ABB RAPID module: Module1.mod

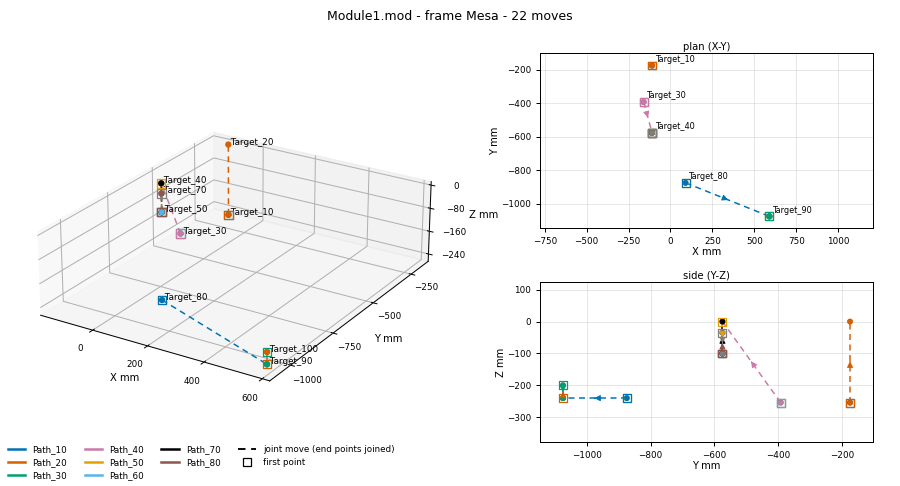
[picture p0: tool path of Module1.mod in frame Mesa, 22 of 23 moves have a stored position in this frame; points joined in program order, loops and branches not executed]
MODULE Module1
    CONST robtarget Target_10:=[[-110,-175,-254],[0.990340804,0,0,-0.138654579],[0,-2,0,0],[9E+09,9E+09,9E+09,9E+09,9E+09,9E+09]];
    CONST robtarget Target_20:=[[-110,-175,0],[0.990340804,0,0,-0.138654579],[0,-2,0,0],[9E+09,9E+09,9E+09,9E+09,9E+09,9E+09]];
    CONST robtarget Target_30:=[[-160,-392.5,-253.927],[1,0,0,0],[0,-2,0,0],[9E+09,9E+09,9E+09,9E+09,9E+09,9E+09]];
    CONST robtarget Target_40:=[[-110,-575,0],[0.990340804,0,0,0.138654579],[0,-2,0,0],[9E+09,9E+09,9E+09,9E+09,9E+09,9E+09]];
    CONST robtarget Target_50:=[[-110,-575,-100],[0.990340804,0,0,0.138654579],[0,-2,0,0],[9E+09,9E+09,9E+09,9E+09,9E+09,9E+09]];
    CONST robtarget Target_60:=[[-110,-575,-100],[0,0.990340804,0.138654579,0],[0,-2,0,0],[9E+09,9E+09,9E+09,9E+09,9E+09,9E+09]];
    CONST robtarget Target_70:=[[-110,-575,-35],[0,0.990340804,0.138654579,0],[0,-2,0,0],[9E+09,9E+09,9E+09,9E+09,9E+09,9E+09]];
    CONST robtarget Target_80:=[[90,-875,-240],[0.923879533,0,0,0.382683432],[0,-2,0,0],[9E+09,9E+09,9E+09,9E+09,9E+09,9E+09]];
    CONST robtarget Target_90:=[[590,-1075,-240],[0.707106781,0,0,0.707106781],[0,-2,0,0],[9E+09,9E+09,9E+09,9E+09,9E+09,9E+09]];
    CONST robtarget Target_100:=[[590,-1075,-200],[0.707106781,0,0,0.707106781],[0,-2,0,0],[9E+09,9E+09,9E+09,9E+09,9E+09,9E+09]];
    CONST robtarget Home:=[[515,0,712],[0.707106781,0,0.707106781,0],[0,-2,0,0],[9E+09,9E+09,9E+09,9E+09,9E+09,9E+09]];
!***********************************************************
    !
    ! M?dulo:  Module1
    !
    ! Descripción:
    !   <Introduzca la descripción aquí>
    !
    ! Autor: acer
    !
    ! Versión: 1.0
    !
    !***********************************************************


    !***********************************************************
    !
    ! Procedimiento Main
    !
    !   Este es el punto de entrada de su programa
    !
    !***********************************************************
    PROC main()
        WHILE TRUE DO
            Path_140;
            IF DI_01 = 1 THEN
                Set DO_01;
                Path_10;
                Set DO_04;
                Reset DO_04;
                WaitTime 0.5;
                Path_20;
                WaitTime 0.5;
                Set DO_05;
                Reset DO_05;
                Set Attach;
                Reset Attach;
                WaitTime 0.5;
                Path_10;
                Path_30;
                Path_40;
                WaitTime 0.5;
                Set DO_04;
                Reset DO_04;
                WaitTime 0.5;
                Set Dettach;
                Reset Dettach;
                Path_50;
                WaitTime 1;
                Path_70;
                WaitTime 0.5;
                Set DO_05;
                Reset DO_05;
                WaitTime 1;
                Set Attach;
                Reset Attach;
                Path_50;
                Path_60;
                Path_80;
                WaitTime 0.5;
                Set DO_04;
                Reset DO_04;
                WaitTime 0.5;
                Set Dettach;
                Reset Dettach;
                Path_90;
                WaitTime 5;
                Path_80;
                WaitTime 1;
                Set DO_05;
                Reset DO_05;
                Set Attach;
                Reset Attach;
                WaitTime 0.5;
                Path_100;
                Path_110;
                Path_120;
                WaitTime 0.5;
                Set DO_04;
                Reset DO_04;
                WaitTime 0.5;
                Set Dettach;
                Reset Dettach;
                Path_130;
                WaitTime 0.5;
                Set DO_05;
                Reset DO_05;
                Path_100;
                Path_30;
                Reset DO_01;
            ENDIF
        ENDWHILE
    ENDPROC

    PROC Path_10()
        MoveJ Target_10,v100,z10,Griper\WObj:=Mesa;
    ENDPROC

    PROC Path_20()
        MoveJ Target_10,v100,z10,Griper\WObj:=Mesa;
        MoveJ Target_20,v100,z10,Griper\WObj:=Mesa;
    ENDPROC
    PROC Path_30()
        MoveJ Target_30,v100,z10,Griper\WObj:=Mesa;
    ENDPROC
    PROC Path_40()
        MoveJ Target_30,v100,z10,Griper\WObj:=Mesa;
        MoveJ Target_40,v100,z10,Griper\WObj:=Mesa;
    ENDPROC
    PROC Path_50()
        MoveJ Target_40,v100,z10,Griper\WObj:=Mesa;
        MoveJ Target_50,v100,z10,Griper\WObj:=Mesa;
    ENDPROC
    PROC Path_60()
        MoveJ Target_60,v100,z100,Griper\WObj:=Mesa;
    ENDPROC
    PROC Path_70()
        MoveJ Target_50,v100,z10,Griper\WObj:=Mesa;
        MoveJ Target_40,v100,z10,Griper\WObj:=Mesa;
    ENDPROC
    PROC Path_80()
        MoveJ Target_60,v100,z10,Griper\WObj:=Mesa;
        MoveJ Target_70,v100,z10,Griper\WObj:=Mesa;
    ENDPROC
    PROC Path_90()
        MoveJ Target_70,v100,z10,Griper\WObj:=Mesa;
        MoveJ Target_60,v100,z10,Griper\WObj:=Mesa;
    ENDPROC
    PROC Path_100()
        MoveJ Target_80,v100,z10,Griper\WObj:=Mesa;
    ENDPROC
    PROC Path_110()
        MoveJ Target_80,v100,z10,Griper\WObj:=Mesa;
        MoveJ Target_90,v100,z10,Griper\WObj:=Mesa;
    ENDPROC
    PROC Path_120()
        MoveJ Target_90,v100,z10,Griper\WObj:=Mesa;
        MoveJ Target_100,v100,z10,Griper\WObj:=Mesa;
    ENDPROC
    PROC Path_130()
        MoveJ Target_100,v100,z10,Griper\WObj:=Mesa;
        MoveJ Target_90,v100,z10,Griper\WObj:=Mesa;
    ENDPROC
    PROC Path_140()
        MoveJ Home,v100,z10,tool0\WObj:=wobj0;
    ENDPROC
ENDMODULE
